TYPE Test_Log :
STRUCT
	Index : INT;
	Description : STRING(255);
	Result : STRING(10);
END_STRUCT
END_TYPE

(* stored: Version 1.1.0.1, ProductVersion 3.1.4024.10
   DUT Test_Log: Id {a80bcfb5-bd0b-4a56-b0c3-ba85d0633d99} *)
